FUNCTION_BLOCK GPIO_controller (* Simple FB with one algorithm *)
  (* Standard: 61499-1 *)
  (* Version 1.0, 2025-07-17, felix *)
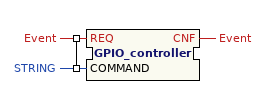
  EVENT_INPUT
    REQ WITH COMMAND; (* Normal Execution Request *)
  END_EVENT
  EVENT_OUTPUT
    CNF; (* Execution Confirmation *)
  END_EVENT
  VAR_INPUT
    COMMAND : STRING;
  END_VAR
  EC_STATES
    REQ : REQ -> CNF;
  END_STATES
  ALGORITHM Req IN ST:

  END_ALGORITHM
END_FUNCTION_BLOCK
